(* CODESYS project MID_IO_Demo.project

Project tree, tasks and I/O mapping:
  Device : Changsha Xiangji-ARM Cortex A9(xilinx zynq7000)-linux, Changsha Xiangji Hiden Technology Co.Ltd, version 3.5.10.20
    application Application
      libraries: Standard, * (System)
      task MainTask (cyclic, interval 4 ms, priority 1) calls PLC_PRG
      task VISU_TASK (cyclic, interval 20 ms, priority 20) calls VisuElems.Visu_Prg
      program PLC_PRG [ST]
      visualisation IO_Demo_Visua
      image pool ImagePool
      global variables GVL
    SoftMotion General Axis Pool
    IoDrvMID7B : IoDrvMID7B, Cyber-MI, version 19.5.1
        input  Application.GVL.AI_00_test : DWORD  // Ai00@P13
        input  Application.GVL.AI_01_test : DWORD  // Ai01@P02
        input  Application.GVL.AI_02_test : DWORD  // Ai02@P01
        input  Application.GVL.AI_03_test : DWORD  // Ai03@P03
        input  Application.GVL.AI_04_test : DWORD  // Ai04@P06
        input  Application.GVL.AI_05_test : DWORD  // Ai05@P05
        input  Application.GVL.AI_06_test : DWORD  // Ai06@P04
        input  Application.GVL.AI_07_test : DWORD  // Ai07@P07
        input  Application.GVL.AI_08_test : DWORD  // Ai08@P35
        input  Application.GVL.AI_09_test : DWORD  // Ai09@P34
        input  Application.GVL.AI_10_test : DWORD  // Ai10@P33
        input  Application.GVL.AI_11_test : DWORD  // Ai11@P32
        input  Application.GVL.AI_12_test : DWORD  // Ai12@P31
        input  Application.GVL.AI_13_test : DWORD  // Ai13@P30
        input  Application.GVL.AI_14_test : DWORD  // Ai14@P29
        input  Application.GVL.AI_15_test : DWORD  // Ai15@P28
        input  Application.GVL.DI_00_test : BOOL  // Di00@P13
        input  Application.GVL.DI_01_test : BOOL  // Di01@P02
        input  Application.GVL.DI_02_test : BOOL  // Di02@P01
        input  Application.GVL.DI_03_test : BOOL  // Di03@P03
        input  Application.GVL.DI_04_test : BOOL  // Di04@P06
        input  Application.GVL.DI_05_test : BOOL  // Di05@P05
        input  Application.GVL.DI_06_test : BOOL  // Di06@P04
        input  Application.GVL.DI_07_test : BOOL  // Di07@P07
        input  Application.GVL.DI_08_test : BOOL  // Di08@P35
        input  Application.GVL.DI_09_test : BOOL  // Di09@P34
        input  Application.GVL.DI_10_test : BOOL  // Di10@P33
        input  Application.GVL.DI_11_test : BOOL  // Di11@P32
        input  Application.GVL.DI_12_test : BOOL  // Di12@P31
        input  Application.GVL.DI_13_test : BOOL  // Di13@P30
        input  Application.GVL.DI_14_test : BOOL  // Di14@P29
        input  Application.GVL.DI_15_test : BOOL  // Di15@P28
        input  Application.GVL.DI_16_test : BOOL  // Di16@P19
        input  Application.GVL.DI_17_test : BOOL  // Di17@P18
        input  Application.GVL.DI_18_test : BOOL  // Di18@P17
        input  Application.GVL.DI_19_test : BOOL  // Di19@P16
        input  Application.GVL.DI_20_test : BOOL  // Di20@P27
        input  Application.GVL.DI_21_test : BOOL  // Di21@P26
        input  Application.GVL.DI_22_test : BOOL  // Di22@14
        input  Application.GVL.PI_00_test : DWORD  // Pi00@P19
        input  Application.GVL.PI_01_test : DWORD  // Pi01@P18
        input  Application.GVL.PI_02_test : DWORD  // Pi02@P26
        input  Application.GVL.PI_03_test : DWORD  // Pi03@P14
        output Application.GVL.DO_00_test : BOOL  // Do00-Ai08@P35
        output Application.GVL.DO_01_test : BOOL  // Do01-Ai09@P34
        output Application.GVL.DO_02_test : BOOL  // Do02-Ai10@P33
        output Application.GVL.DO_03_test : BOOL  // Do03-Ai11@P32
        output Application.GVL.DO_04_test : BOOL  // Do04-Ai12@P31
        output Application.GVL.DO_05_test : BOOL  // Do05-Ai13@P30
        output Application.GVL.DO_06_test : BOOL  // Do06-Ai14@P29
        output Application.GVL.DO_07_test : BOOL  // Do07-Ai15@P28
        output Application.GVL.PWM_00_test : DWORD  // PWM00@P33
        output Application.GVL.PWM_01_test : DWORD  // PWM01@P32
        output Application.GVL.PWM_02_test : DWORD  // PWM02@P31
        output Application.GVL.PWM_03_test : DWORD  // PWM03@P30
        output Application.GVL.PWM_04_test : DWORD  // PWM04@P29
        output Application.GVL.PWM_05_test : DWORD  // PWM05@P28
        unmapped channels: Ai16, Ai17, Ai18, Ai19, Ai20, Ai21, Ai22, Ai23, Di23, Di24, Di25, Di26, Di27, Di28, Di29, Di30, Di31, Pi04@P19-18-17, Pi05@P16-27-26, Pi06, Pi07, PWM06, PWM07
  libraries: VisuSymbols, 3.5.10.0 (System)
  text list GlobalTextList
  5ce3da45-db07-42e7-a21c-a00fff4ed8f6|companyLOG.jpg
*)

// Device/Application/GVL
{attribute 'qualified_only'}
{attribute 'qualified_only'}


VAR_GLOBAL
	AI_00_test:DWORD;
    AI_01_test:DWORD;
    AI_02_test:DWORD;
    AI_03_test:DWORD;
    AI_04_test:DWORD;
    AI_05_test:DWORD;
    AI_06_test:DWORD;
    AI_07_test:DWORD;
    AI_08_test:DWORD;
    AI_09_test:DWORD;
    AI_10_test:DWORD;
    AI_11_test:DWORD;
    AI_12_test:DWORD;
    AI_13_test:DWORD;
    AI_14_test:DWORD;
    AI_15_test:DWORD;
	
	DI_00_test:BOOL;
    DI_01_test:BOOL;
    DI_02_test:BOOL;
    DI_03_test:BOOL;
    DI_04_test:BOOL;
    DI_05_test:BOOL;
    DI_06_test:BOOL;
    DI_07_test:BOOL;
    DI_08_test:BOOL;
    DI_09_test:BOOL;
    DI_10_test:BOOL;
    DI_11_test:BOOL;
    DI_12_test:BOOL;
    DI_13_test:BOOL;
    DI_14_test:BOOL;
    DI_15_test:BOOL;
    DI_16_test:BOOL;
    DI_17_test:BOOL;
    DI_18_test:BOOL;
    DI_19_test:BOOL;
    DI_20_test:BOOL;
    DI_21_test:BOOL;
    DI_22_test:BOOL;

	PI_00_test:DWORD;
	PI_01_test:DWORD;
	PI_02_test:DWORD;
	PI_03_test:DWORD;
	
	DO_00_test:BOOL;
    DO_01_test:BOOL;
    DO_02_test:BOOL;
    DO_03_test:BOOL;
    DO_04_test:BOOL;
    DO_05_test:BOOL;
    DO_06_test:BOOL;
    DO_07_test:BOOL;
	
	PWM_00_test:DWORD;
    PWM_01_test:DWORD;
    PWM_02_test:DWORD;
    PWM_03_test:DWORD;
    PWM_04_test:DWORD;
    PWM_05_test:DWORD;
	
	PWMI_00_test:DWORD;
	PWMI_01_test:DWORD;
	PWMI_02_test:DWORD;
	PWMI_03_test:DWORD;
	

	
END_VAR

// Device/Application/PLC_PRG
PROGRAM PLC_PRG
VAR
	
	ton1:TON;
	AI00_TempValue:REAL;
    AI00_Temp:DWORD;
	AI00_Min:DWORD:=30000;
	AI00_Max:DWORD:=0;
	AI00_Avr:REAL:=0;
	AI00_AvrValue:REAL;
	AI_TEST_NUM: DWORD:=0;

	
END_VAR



//使用DO-00端口控制一个指示灯（一个程序周期闪一次）
     GVL.DO_00_TEST:=NOT GVL.DO_00_TEST;
	 
//使用一个DO-01端口控制一个指示灯（一秒钟闪一次）
TON1(IN:=TRUE,PT:=T#1S);
IF TON1.Q=TRUE THEN
   GVL.DO_01_TEST:=NOT GVL.DO_01_TEST;
   TON1(IN:=FALSE,PT:=T#1S);
END_IF

//监测一个DI端口，当输入为高时，控制一个DO端口的输出24V,否则不输出
IF GVL.DI_00_TEST THEN
   GVL.DO_03_TEST:=TRUE;
ELSE
   GVL.DO_03_TEST:=FALSE;
END_IF

//取AI-00采集到的瞬态值、最小值、平均值和最大值
AI00_TempValue:=ANY_TO_REAL(GVL.AI_00_TEST)/1000;//AI 端口采集到的瞬态电压值，单位V，采集范围0-24V；
AI00_Temp:=GVL.AI_00_TEST;

IF AI_TEST_NUM<=10 THEN                          //每次采20个数取最小值、最大值和 平均值 
	AI_TEST_NUM:=AI_TEST_NUM+1;
         IF  AI00_min> AI00_temp THEN
			 AI00_min:= AI00_temp;
		 END_IF
		 
		 IF  AI00_max< AI00_temp THEN
			 AI00_max:= AI00_temp;
		 END_IF
		 
		  IF  AI00_avr=0  THEN
			  AI00_avr:=(ANY_TO_REAL(AI00_max)+ANY_TO_REAL(AI00_min))/2;
		  ELSE
			 AI00_Avr:= AI00_Avr*0.99+ ANY_TO_REAL(AI00_temp)*0.01;
		  END_IF
ELSE
	AI00_min:=30000;
	AI00_max:=0;
	AI00_avr:=0;
	AI_TEST_NUM:=0;
END_IF

END_PROGRAM

// Device/Application/IO_Demo_Visua
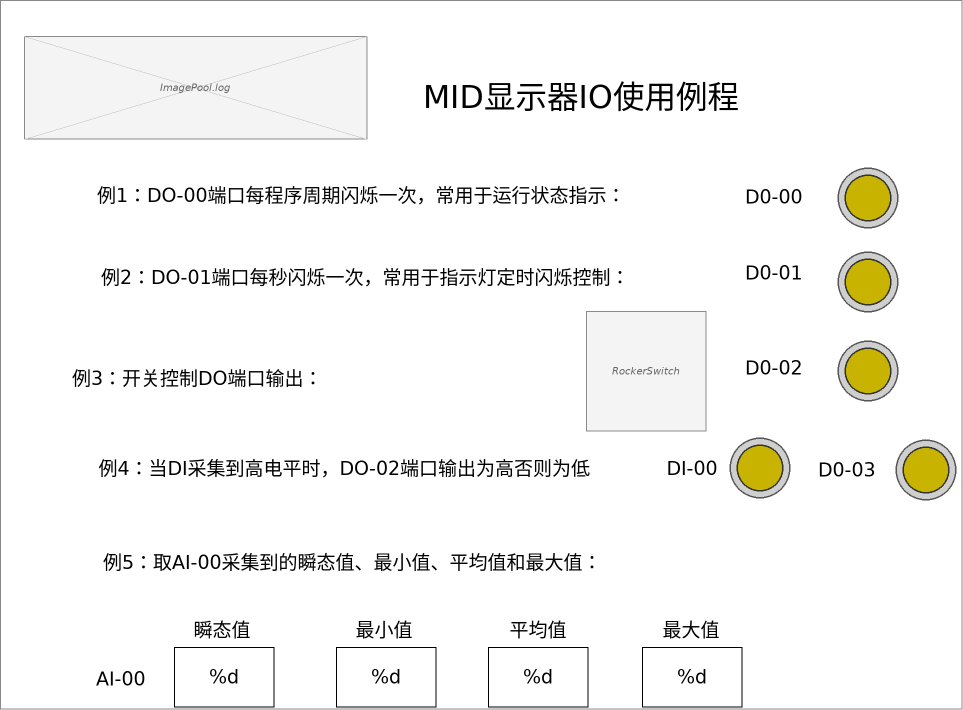
VISUALIZATION IO_Demo_Visua  // 963x710
    Label (294,54 574x86), "MID显示器IO使用例程"
    RockerSwitch (586,311 120x120), variable: GVL.DO_02_test, behaviour: TOGGLE, style: Switch-RockerSwitch-Gray
    Label (44,535 617x55), "例5：取AI-00采集到的瞬态值、最小值、平均值和最大值："
    Label (744,167 60x60), "D0-00"
    Label (172,600 100x60), "瞬态值"
    Rectangle (174,647 100x60), "%d", text variable: PLC_PRG.AI00_Temp
    Label (36,168 651x55), "例1：DO-00端口每程序周期闪烁一次，常用于运行状态指示："
    Label (24,250 683x55), "例2：DO-01端口每秒闪烁一次，常用于指示灯定时闪烁控制："
    Label (744,243 60x60), "D0-01"
    Label (20,441 649x55), "例4：当DI采集到高电平时，DO-02端口输出为高否则为低"
    Label (638,443 108x51), "DI-00"
    Label (819,440 56x60), "D0-03"
    Label (334,600 100x60), "最小值"
    Rectangle (336,647 100x60), "%d", text variable: PLC_PRG.AI00_Min
    Label (488,600 100x60), "平均值"
    Rectangle (488,647 100x60), "%d", text variable: PLC_PRG.AI00_Avr
    Label (641,600 100x60), "最大值"
    Rectangle (642,647 100x60), "%d", text variable: PLC_PRG.AI00_Max
    Label (71,650 100x58), "AI-00"
    Label (30,351 335x55), "例3：开关控制DO端口输出："
    Lamp1 (833,163 70x70), variable: GVL.DO_00_test, style: Lamp-Lamp1-Yellow
    Lamp1 (833,247 70x70), variable: GVL.DO_01_test, style: Lamp-Lamp1-Yellow
    Lamp1 (725,433 70x70), variable: GVL.DI_00_test, style: Lamp-Lamp1-Yellow
    Lamp1 (891,435 70x70), variable: GVL.DO_03_test, style: Lamp-Lamp1-Yellow
    Lamp1 (833,336 70x70), variable: GVL.DO_02_test, style: Lamp-Lamp1-Yellow
    Label (744,338 60x60), "D0-02"
    Image (24,36 343x103), image: ImagePool.log
END_VISUALIZATION
